Staubli VAL3: cmdShutdown.pgx

public program cmdShutdown(num& x_nAxNum)
begin
  //关闭指定驱动器，设置"switch on"为false
  //shutdown的顺序参考相应电机说明
  doFaultReset[x_nAxNum]=false
  doQuickStop[x_nAxNum]=true
  doEnableVoltage[x_nAxNum]=true
  doSwitchOn[x_nAxNum]=false
  delay(0.004)
end
